Staubli VAL3: interfaceCS9.pjx

--- interfaceCS9.pjx ---
Parameters version=s7.11 stackSize=5000 millimeterUnit=true
Program file=ack.pgx
Program file=cartStatus.pgx
Program file=clearScreen.pgx
Program file=debug.pgx
Program file=feedbackStatus.pgx
Program file=init.pgx
Program file=motionBuffer.pgx
Program file=motionProgress.pgx
Program file=motionStatus.pgx
Program file=start.pgx
Program file=stop.pgx
Program file=trajBuffer.pgx
Program file=velOverwrite.pgx
Data file=interfaceCS9.dtx
Library alias=libQueueFuncs path=Disk://ros_libs/QueueFuncs/QueueFuncs.pjx

--- cartStatus.pgx ---
public program cartStatus(num x_nCartConnFlag, num x_nLastMsgAge)
begin

  // update cartesian status on port 11001

  switch x_nCartConnFlag
    case -1
      userPageSet("uxMonitor", "lblCartState", "innerHTML", "connection lost")
    break
    case 0
      userPageSet("uxMonitor", "lblCartState", "innerHTML", "not connected")
    break
    case 1
      userPageSet("uxMonitor", "lblCartState", "innerHTML", "connected")
    break
    default
      userPageSet("uxMonitor", "lblCartState", "innerHTML", "not connected")
    break
  endSwitch

  if (x_nLastMsgAge < 0)
    userPageSet("uxMonitor", "lblCartAge", "innerHTML", "last msg: n/a")
  else
    userPageSet("uxMonitor", "lblCartAge", "innerHTML", "last msg: " + toString(".1", x_nLastMsgAge) + " s")
  endIf

end
